FUNCTION_BLOCK FB_Sum
VAR_INPUT
	one : UINT;
    two : UINT;
END_VAR
VAR_OUTPUT
    result : UINT;
END_VAR
VAR
	_prop:BOOL:=FALSE;
END_VAR

PROPERTY Prop : BOOL
GET
Prop := _prop;
END_GET
SET
_prop:=Prop;
END_SET
END_PROPERTY

END_FUNCTION_BLOCK

(* stored: Version 1.1.0.1, ProductVersion 3.1.4024.12
   POU FB_Sum: Id {5173c1cb-3f1b-4feb-a554-e8293792cdc5}, SpecialFunc None
   Property Prop: Id {2a6005bf-f31a-4407-98c1-15d61d1ba5ea}
   Get Get: Id {30a238ee-ef8c-4c1e-88d2-d2570e70303e}
   Set Set: Id {256b49a1-362a-4142-9c27-521044afa2d5} *)
